Staubli VAL3: powerSwitch.pgx

program powerSwitch(bool enable (dimensions=1), string command (dimensions=1), num sio_ID (dimensions=1))
  local string reply
begin
  //**************************************************
  // Method to enable or disable the power on the robot, depending whether the
  // enable variable is true or false. Command argument is needed to construct
  // the reply
  //**************************************************
  if enable
    enablePower()
  else
    disablePower()
  endIf

  if (watch(isPowered()==enable,5)==false)
    reply=command+":fail_'RobotPowerCannotBeSwitched'"
  else
    reply=command+":done"
  endIf
  taskCreate "sendStatus",10,sendStatus(reply,sio_ID)
  taskKill("powerSwitch")
end
